// TIA Portal V20 program export: 0 tag tables, 0 data types, 3 data blocks, 3 code blocks (in call order from the OBs), 0 instance data blocks

DATA_BLOCK "Dati"
{ S7_Optimized_Access := 'TRUE' }
VERSION : 0.1
NON_RETAIN
   VAR 
      in1 : Bool;
      out1 : Bool;
      in2 : Bool;
      out2 : Bool;
      alarm : Bool;
      alarm2 : Bool;
   END_VAR


BEGIN

END_DATA_BLOCK

DATA_BLOCK "FB_NEW_DB"
{ S7_Optimized_Access := 'TRUE' }
VERSION : 0.1
NON_RETAIN
"FB_NEW"

BEGIN

END_DATA_BLOCK

DATA_BLOCK "FB_NEW_DB_1"
{ S7_Optimized_Access := 'TRUE' }
VERSION : 0.1
NON_RETAIN
"FB_NEW"

BEGIN

END_DATA_BLOCK

ORGANIZATION_BLOCK "Main"   // OB1, LAD, ProgramCycle
TITLE = "Main Program Sweep (Cycle)"
{ S7_Optimized_Access := 'TRUE' }
// stored: SetENOAutomatically false
   VAR_INPUT
      Initial_Call : Bool;   // Initial call of this OB
      Remanence : Bool;   // =True, if remanent data are available
   END_VAR
BEGIN

REGION Network 1
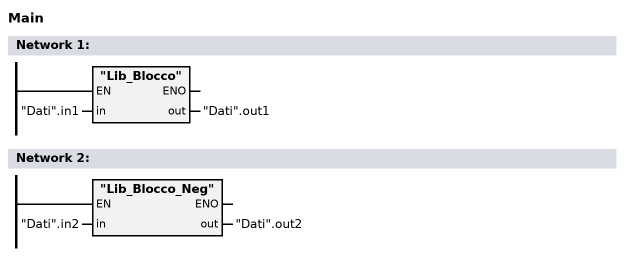
   RUNG wire#powerrail
      "Lib_Blocco"(in := "Dati".in1, out => "Dati".out1)
   END_RUNG
   // the same network as SCL:
   "Lib_Blocco"(in := "Dati".in1, out => "Dati".out1);
END_REGION

REGION Network 2
   RUNG wire#powerrail
      "Lib_Blocco_Neg"(in := "Dati".in2, out => "Dati".out2)
   END_RUNG
   // the same network as SCL:
   "Lib_Blocco_Neg"(in := "Dati".in2, out => "Dati".out2);
END_REGION
END_ORGANIZATION_BLOCK

FUNCTION_BLOCK "FB_NEW"   // FB2, LAD
{ S7_Optimized_Access := 'TRUE' }
// stored: MemoryReserve 100, SetENOAutomatically false
   VAR_INPUT
      in : Bool;
   END_VAR
   VAR_OUTPUT
      out : Bool;
   END_VAR
BEGIN

REGION Network 1
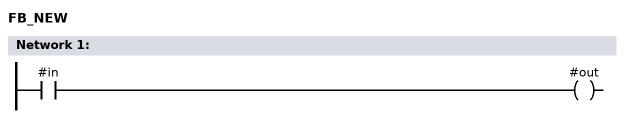
   RUNG wire#powerrail
      Contact( #in )
      Coil( #out )
   END_RUNG
   // the same network as SCL:
   #out := #in;
END_REGION
END_FUNCTION_BLOCK

ORGANIZATION_BLOCK "Main_1"
TITLE = "Main Program Sweep (Cycle)"
{ S7_Optimized_Access := 'TRUE' }
VERSION : 0.1

BEGIN
	"FB_NEW_DB_1"(in:=false);
	
END_ORGANIZATION_BLOCK
